{attribute 'GeneratedUsingTerminal: EL3632-0000-0016'}
{attribute addProperty BoxType "EL3632-0000-0016"}
{attribute addProperty Id "Ch1_ValueAT %I*INT2"}
{attribute addProperty CRC "2803750145"}
{attribute addProperty Size "2"}
TYPE Ch1_Sample_A71DD501 EXTENDS InputBase_8311D824 :
STRUCT
	{attribute addProperty Name "Ch1_Value"}
	Ch1_Value AT %I* : INT;
END_STRUCT
END_TYPE

(* stored: Version 1.2.0.0, ProductVersion 3.1.4024.11
   DUT Ch1_Sample_A71DD501: Id {c84d9180-b10a-4855-8a99-3d715d100cb2} *)
